INTERFACE I_WritableData

PROPERTY PUBLIC Data : T_MAXSTRING
GET
END_GET
END_PROPERTY

METHOD PUBLIC TrySet : BOOL;
VAR_INPUT
	Value : ANY;
END_VAR
END_METHOD

METHOD PUBLIC TrySetFrom : BOOL;
VAR_INPUT
	SourceAddress : PVOID;
	SourceSize : UDINT;
END_VAR
END_METHOD

END_INTERFACE

(* stored: Version 1.1.0.1, ProductVersion 3.1.4024.12
   Itf I_WritableData: Id {87191d5d-b323-4120-9c02-78646e324ac0}
   Property Data: Id {dbdae43e-426a-4e2b-935f-e004162b6789}
   Get Get: Id {5b9672d7-9010-4de1-a1cc-cf895596a18b}
   Method TrySet: Id {b17c43ca-c04d-4614-b0c8-b76a7cfcbe9b}
   Method TrySetFrom: Id {8ec144fc-c13e-419b-82d9-eb5b19b9b209} *)
